// TIA Portal project "height_sorting" (V16)
// Vorlageprojekt für das Buch mit Zielsystem S7-1200

(* hardware
DEVICE "S7-1200-Station_1"  S7-1200 Station
   slot 0: "Baugruppenträger_0"  Rack  V1.0
   slot 1: "PLC_1"  CPU 1211C DC/DC/DC  6ES7 211-1AE40-0XB0  V4.1
*)

// ===== PLC "PLC_1"  CPU 1211C DC/DC/DC =====

VAR_GLOBAL   // PLC tag table "Standard-Variablentabelle"
   "feeder conveyor" AT %A0.0 : Bool;
   "optical entry" AT %E0.0 : Bool;
   "opt low box" AT %E0.1 : Bool;
   "Start" AT %I1.3 : Bool;
   "Stop" AT %I1.5 : Bool;
   "Start/Stop" AT %M0.0 : Bool;
   "entry conveyor" AT %Q0.1 : Bool;
   "back proximity" AT %I0.5 : Bool;
   "front proximity" AT %I0.6 : Bool;
   "turn motor" AT %Q0.4 : Bool;
   "turntable entry" AT %I0.3 : Bool;
   "load conveyor" AT %Q0.2 : Bool;
   "Storage Byte" AT %MB10 : Byte;
   "Tag_1" AT %M0.1 : Bool;
   "opt high box" AT %I0.2 : Bool;
   "decision bit" AT %M10.0 : Bool;
   "shifted bit" AT %M10.2 : Bool;
   "unload conveyor" AT %Q0.3 : Bool;
   "Totally rotated" AT %M0.2 : Bool;
   "right conveyor" AT %Q0.6 : Bool;
   "left coveyor" AT %Q0.5 : Bool;
   "opt end right" AT %I1.1 : Bool;
   "Tag_4" AT %M0.4 : Bool;
   "opt end left" AT %I1.2 : Bool;
   "Tag_6" AT %M0.5 : Bool;
   "opt end right conv neg" AT %M0.6 : Bool;
   "opt end left conv neg" AT %M0.7 : Bool;
   "opt right entry" AT %I0.7 : Bool;
   "Tag_5" AT %M1.0 : Bool;
   "opt left entry" AT %I1.0 : Bool;
   "Tag_7" AT %M1.2 : Bool;
   "opt right neg" AT %M1.1 : Bool;
   "opt left neg" AT %M1.3 : Bool;
   "Tag_2" AT %M1.4 : Bool;
   "digital display" AT %QD30 : DWord;
   "reset button" AT %I1.4 : Bool;
   "Tag_3" AT %M1.5 : Bool;
   "Tag_8" AT %M1.7 : Bool;
   "right box memory" AT %M1.6 : Bool;
   "left box memory" AT %M2.0 : Bool;
END_VAR

// folder: System blocks/Program resources

DATA_BLOCK "Timer1"   // DB1
{ S7_Optimized_Access := 'TRUE' }
AUTHOR : Simatic
FAMILY : IEC
NAME : IEC_TMR
VERSION : 1.0
// stored: InstanceOfName IEC_TIMER
"IEC_TIMER"
BEGIN
END_DATA_BLOCK

DATA_BLOCK "C1"   // DB2
{ S7_Optimized_Access := 'TRUE' }
AUTHOR : Simatic
FAMILY : IEC
NAME : CNTR
VERSION : 1.0
// stored: InstanceOfName IEC_COUNTER
"IEC_COUNTER"
BEGIN
END_DATA_BLOCK

DATA_BLOCK "C2"   // DB3
{ S7_Optimized_Access := 'TRUE' }
AUTHOR : Simatic
FAMILY : IEC
NAME : CNTR
VERSION : 1.0
// stored: InstanceOfName IEC_COUNTER
"IEC_COUNTER"
BEGIN
END_DATA_BLOCK

DATA_BLOCK "C3"   // DB4
{ S7_Optimized_Access := 'TRUE' }
AUTHOR : Simatic
FAMILY : IEC
NAME : CNTR
VERSION : 1.0
// stored: InstanceOfName IEC_COUNTER
"IEC_COUNTER"
BEGIN
END_DATA_BLOCK

// folder: (top level)

FUNCTION "MHJ-PLC-Lab-Function-S71200" : Void   // FC9000, SCL
{ S7_Optimized_Access := 'TRUE' }
VERSION : 0.1
   VAR_TEMP
      rdTimeReturn : Int;
      outputTime : DTL;
      SyncVal : Byte;
      forVal : Int;
      forVal_2 : Int;
      Value : Byte;
   END_VAR
   VAR CONSTANT
      CompVal : Byte := 16#34;
      Value_01 : Byte := 16#11;
      Value_01_DW : DWord := 16#A165_D992;
      Value_02_DW : DWord := 16#58BE_4401;
   END_VAR
BEGIN

   #Value:=PEEK(area := 16#82,
        dbNumber := 0,
        byteOffset := 511);
   #Value := #Value + 1;

   POKE(area := 16#82,
        dbNumber := 0,
        byteOffset := 511,
        value := #Value);

   POKE(area:=16#81,
        dbNumber:=0,
        byteOffset:=1016,
        value:=#Value_01_DW);
   POKE(area := 16#81,
        dbNumber := 0,
        byteOffset := 1020,
        value := #Value_02_DW);

   POKE(area := 16#81,
        dbNumber := 0,
        byteOffset := 511,
        value := B#16#00);

   FOR #forVal := 0 TO 120 DO
       FOR #forVal_2:=0 TO 10 DO
           #rdTimeReturn:=RD_SYS_T(#outputTime);
           #rdTimeReturn := WR_SYS_T(#outputTime);
           #rdTimeReturn := RD_SYS_T(#outputTime);
           #rdTimeReturn := WR_SYS_T(#outputTime);
       END_FOR;
       #SyncVal:= PEEK(area := 16#81,
                      dbNumber := 0,
                      byteOffset := 511);
       IF #SyncVal = #CompVal THEN
          GOTO M_1;
       END_IF;
   END_FOR;
   RETURN;

   M_1:
   POKE(area := 16#81,
        dbNumber := 0,
        byteOffset := 511,
        value := B#16#0);
END_FUNCTION

ORGANIZATION_BLOCK "Main"   // OB1, LAD, ProgramCycle
TITLE = "Main Program Sweep (Cycle)"
{ S7_Optimized_Access := 'TRUE' }
VERSION : 0.1
   VAR_INPUT
      Initial_Call : Bool;   // Initial call of this OB
      Remanence : Bool;   // =True, if remanent data are available
   END_VAR
   VAR_TEMP   // added for the SCL form of the ladder/FBD networks
      _w1 : Bool;
      _w2 : Bool;
      _w3 : Bool;
      _w4 : Bool;
   END_VAR
BEGIN

REGION Network 1: Konnektierungsbaustein für PLC-Lab
   // Im Netzwerk 1 wird der Konnektierungsbaustein für PLC-Lab aufgerufen.
   // Dieser Aufruf darf nicht entfernt werden!
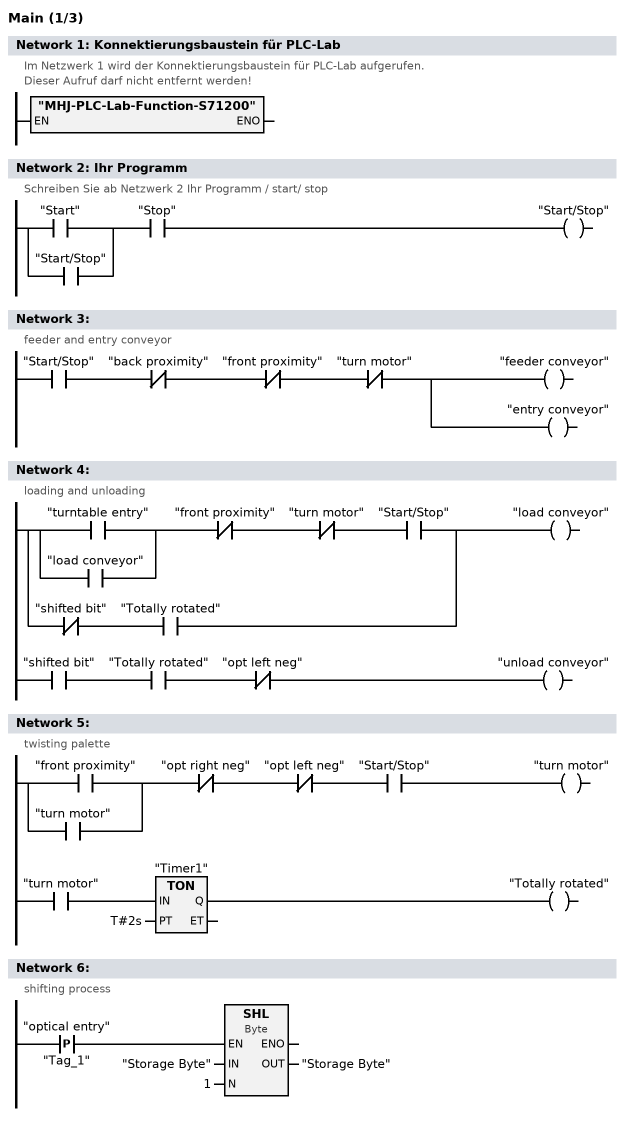
   RUNG wire#powerrail
      "MHJ-PLC-Lab-Function-S71200"()
   END_RUNG
   // the same network as SCL:
   "MHJ-PLC-Lab-Function-S71200"();
END_REGION

REGION Network 2: Ihr Programm
   // Schreiben Sie ab Netzwerk 2 Ihr Programm / start/ stop
   RUNG wire#powerrail
      Contact( "Start" )
      wire#w1
      Contact( "Stop" )
      Coil( "Start/Stop" )
   END_RUNG
   RUNG wire#powerrail
      Contact( "Start/Stop" )
   END_RUNG wire#w1
   // the same network as SCL:
   "Start/Stop" := ("Start" OR "Start/Stop") AND "Stop";
END_REGION

REGION Network 3
   // feeder and entry conveyor
   RUNG wire#powerrail
      Contact( "Start/Stop" )
      I_Contact( "back proximity" )
      I_Contact( "front proximity" )
      I_Contact( "turn motor" )
      wire#w1
      Coil( "feeder conveyor" )
   END_RUNG
   RUNG wire#w1
      Coil( "entry conveyor" )
   END_RUNG
   // the same network as SCL:
   "feeder conveyor" := "Start/Stop" AND NOT "back proximity" AND NOT "front proximity" AND NOT "turn motor";
   "entry conveyor" := "feeder conveyor";
END_REGION

REGION Network 4
   // loading and unloading
   RUNG wire#powerrail
      Contact( "turntable entry" )
      wire#w1
      I_Contact( "front proximity" )
      I_Contact( "turn motor" )
      Contact( "Start/Stop" )
      wire#w2
      Coil( "load conveyor" )
   END_RUNG
   RUNG wire#powerrail
      Contact( "load conveyor" )
   END_RUNG wire#w1
   RUNG wire#powerrail
      I_Contact( "shifted bit" )
      Contact( "Totally rotated" )
   END_RUNG wire#w2
   RUNG wire#powerrail
      Contact( "shifted bit" )
      Contact( "Totally rotated" )
      I_Contact( "opt left neg" )
      Coil( "unload conveyor" )
   END_RUNG
   // the same network as SCL:
   "load conveyor" := (("turntable entry" OR "load conveyor") AND NOT "front proximity" AND NOT "turn motor" AND "Start/Stop") OR (NOT "shifted bit" AND "Totally rotated");
   "unload conveyor" := "shifted bit" AND "Totally rotated" AND NOT "opt left neg";
END_REGION

REGION Network 5
   // twisting palette
   "turn motor" := ("front proximity" OR "turn motor") AND NOT "opt right neg" AND NOT "opt left neg" AND "Start/Stop";
   "Timer1".TON(IN := "turn motor", PT := T#2s);
   "Totally rotated" := "Timer1".Q;
END_REGION

REGION Network 6
   // shifting process
   RUNG wire#powerrail
      P_Contact(operand := "optical entry", bit := "Tag_1")
      { S7_Templates := "SrcType := Byte" } Shl(in := "Storage Byte", n := 1, out => "Storage Byte")
   END_RUNG
   // the same network as SCL:
   #_w1 := "optical entry" AND NOT "Tag_1";   // rising edge of "optical entry"
   "Tag_1" := "optical entry";
   IF #_w1 THEN "Storage Byte" := SHL(IN := "Storage Byte", N := 1); END_IF;
END_REGION

REGION Network 7
   // box type
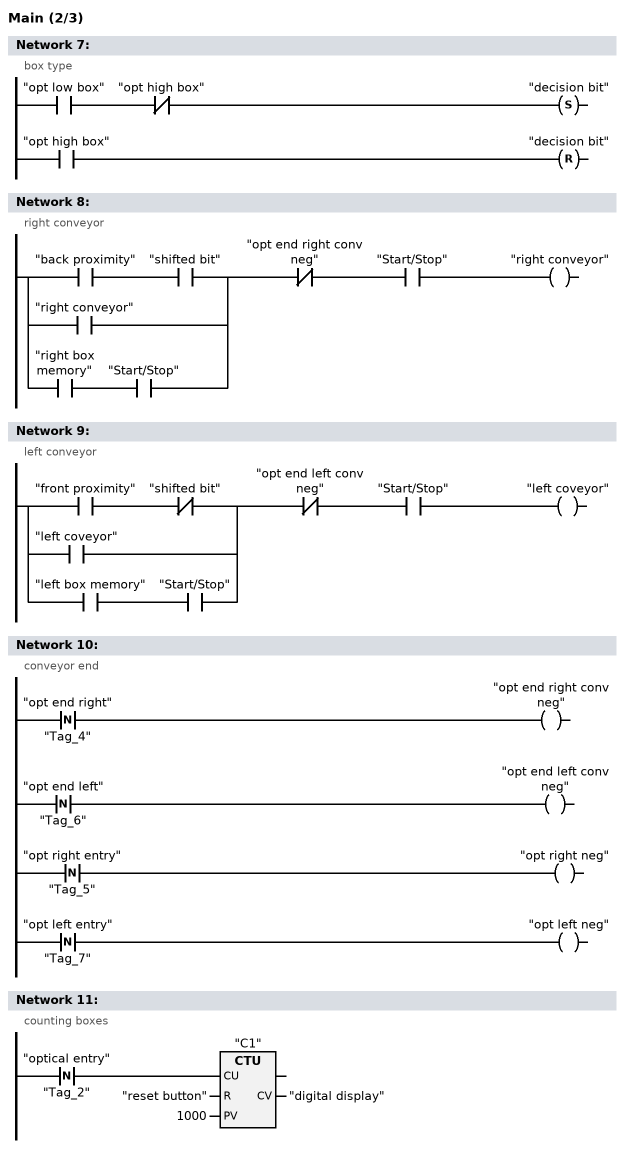
   RUNG wire#powerrail
      Contact( "opt low box" )
      I_Contact( "opt high box" )
      S_Coil( "decision bit" )
   END_RUNG
   RUNG wire#powerrail
      Contact( "opt high box" )
      R_Coil( "decision bit" )
   END_RUNG
   // the same network as SCL:
   IF "opt low box" AND NOT "opt high box" THEN "decision bit" := TRUE; END_IF;
   IF "opt high box" THEN "decision bit" := FALSE; END_IF;
END_REGION

REGION Network 8
   // right conveyor
   RUNG wire#powerrail
      Contact( "back proximity" )
      Contact( "shifted bit" )
      wire#w1
      I_Contact( "opt end right conv neg" )
      Contact( "Start/Stop" )
      Coil( "right conveyor" )
   END_RUNG
   RUNG wire#powerrail
      Contact( "right conveyor" )
   END_RUNG wire#w1
   RUNG wire#powerrail
      Contact( "right box memory" )
      Contact( "Start/Stop" )
   END_RUNG wire#w1
   // the same network as SCL:
   "right conveyor" := (("back proximity" AND "shifted bit") OR "right conveyor" OR ("right box memory" AND "Start/Stop")) AND NOT "opt end right conv neg" AND "Start/Stop";
END_REGION

REGION Network 9
   // left conveyor
   RUNG wire#powerrail
      Contact( "front proximity" )
      I_Contact( "shifted bit" )
      wire#w1
      I_Contact( "opt end left conv neg" )
      Contact( "Start/Stop" )
      Coil( "left coveyor" )
   END_RUNG
   RUNG wire#powerrail
      Contact( "left coveyor" )
   END_RUNG wire#w1
   RUNG wire#powerrail
      Contact( "left box memory" )
      Contact( "Start/Stop" )
   END_RUNG wire#w1
   // the same network as SCL:
   "left coveyor" := (("front proximity" AND NOT "shifted bit") OR "left coveyor" OR ("left box memory" AND "Start/Stop")) AND NOT "opt end left conv neg" AND "Start/Stop";
END_REGION

REGION Network 10
   // conveyor end
   RUNG wire#powerrail
      N_Contact(operand := "opt end right", bit := "Tag_4")
      Coil( "opt end right conv neg" )
   END_RUNG
   RUNG wire#powerrail
      N_Contact(operand := "opt end left", bit := "Tag_6")
      Coil( "opt end left conv neg" )
   END_RUNG
   RUNG wire#powerrail
      N_Contact(operand := "opt right entry", bit := "Tag_5")
      Coil( "opt right neg" )
   END_RUNG
   RUNG wire#powerrail
      N_Contact(operand := "opt left entry", bit := "Tag_7")
      Coil( "opt left neg" )
   END_RUNG
   // the same network as SCL:
   #_w1 := NOT "opt end right" AND "Tag_4";   // falling edge of "opt end right"
   "Tag_4" := "opt end right";
   "opt end right conv neg" := #_w1;
   #_w2 := NOT "opt end left" AND "Tag_6";   // falling edge of "opt end left"
   "Tag_6" := "opt end left";
   "opt end left conv neg" := #_w2;
   #_w3 := NOT "opt right entry" AND "Tag_5";   // falling edge of "opt right entry"
   "Tag_5" := "opt right entry";
   "opt right neg" := #_w3;
   #_w4 := NOT "opt left entry" AND "Tag_7";   // falling edge of "opt left entry"
   "Tag_7" := "opt left entry";
   "opt left neg" := #_w4;
END_REGION

REGION Network 11
   // counting boxes
   #_w1 := NOT "optical entry" AND "Tag_2";   // falling edge of "optical entry"
   "Tag_2" := "optical entry";
   "C1".CTU(CU := #_w1, R := "reset button", PV := 1000, CV => "digital display");
END_REGION

REGION Network 12
   // box memory
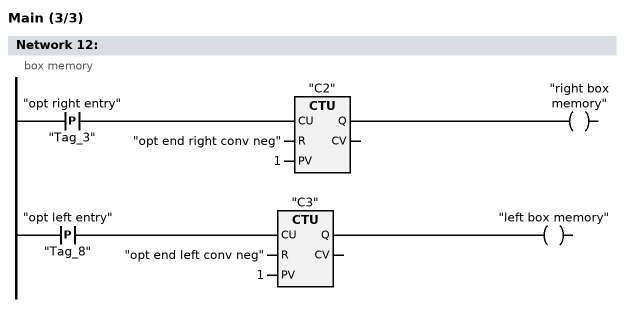
   #_w1 := "opt right entry" AND NOT "Tag_3";   // rising edge of "opt right entry"
   "Tag_3" := "opt right entry";
   "C2".CTU(CU := #_w1, R := "opt end right conv neg", PV := 1);
   "right box memory" := "C2".Q;
   #_w2 := "opt left entry" AND NOT "Tag_8";   // rising edge of "opt left entry"
   "Tag_8" := "opt left entry";
   "C3".CTU(CU := #_w2, R := "opt end left conv neg", PV := 1);
   "left box memory" := "C3".Q;
END_REGION
END_ORGANIZATION_BLOCK

ORGANIZATION_BLOCK "Main_1"   // OB123, LAD, ProgramCycle
TITLE = "Main Program Sweep (Cycle)"
{ S7_Optimized_Access := 'TRUE' }
VERSION : 0.1
   VAR_INPUT
      Initial_Call : Bool;   // Initial call of this OB
      Remanence : Bool;   // =True, if remanent data are available
   END_VAR
BEGIN
END_ORGANIZATION_BLOCK